// TwinCAT 3 PLC project hxr_jjslit_motion
// ProgramVersion: 3.1.4022.7
// libraries:
//   lcls-twincat-motion, * (SLAC)
//   Tc2_Standard, * (Beckhoff Automation GmbH)
//   Tc2_System, * (Beckhoff Automation GmbH)
//   Tc3_Module, * (Beckhoff Automation GmbH)
// project tree:
//   / PlcTask.TcTTO (not stored)
//   POUs/ Main.TcPOU
// real-time tasks:
//   TASK PlcTask: cycle T#10ms, priority 20, ADS port 350
// motion (NC):
//   TASK NC-Task 1 SAF: cycle T#2ms, priority 4, ADS port 501
//   TASK NC-Task 1 SVB: cycle T#10ms, priority 8, ADS port 511
//   AXIS VonHamosY (id 1)
//     Dynamic: AccelerationMaximum=30, DecelerationMaximum=30, Acceleration=14.9254, Deceleration=14.9254, Jerk=44.5534, DelayTime=0.008
//     Velo: RefSearch=0.1, RefSync=0.1, SlowManual=0.1, FastManual=0.2, Maximum=1.5
//     OtherSettings: AllowMotionCmdToSlave=true, PulseDistancePos=0.5, PulseDistanceNeg=0.5
//     encoder EncType=4
//       EncPara: ScaleFactorNumerator=1.5625e-05, Inverse=true, MaxCount=#x0000ffff
//         SoftEndMaxControl: Enable=true, Range=25
//         Inc: RefSoftSyncMask=#x0000ffff
//     drive DrvType=24
//       DrvPara: Inverse=true
//         Analog: VeloReferenz=2, ScaleFactorActTorque=0.1
//         TimeComp: TaskDelayCycles=1
//     controller CtrType=1
//       CtrPara: PriorControlFactor=1
//         PosDiffControl: Range=1
//         Observer: BandWidth=20
//   AXIS Axis 2 (Spare) (id 2)
//     OtherSettings: AllowMotionCmdToSlave=true
//     encoder EncType=4
//       EncPara: MaxCount=#x0000ffff
//         Inc: RefSoftSyncMask=#x0000ffff
//     drive DrvType=24
//       Analog: ScaleFactorActTorque=0.1
//       TimeComp: TaskDelayCycles=1
//     controller CtrType=1
//       CtrPara: PriorControlFactor=1
//         Observer: BandWidth=20
//   AXIS Axis 3 (Spare) (id 3)
//     OtherSettings: AllowMotionCmdToSlave=true
//     encoder EncType=4
//       EncPara: MaxCount=#x0000ffff
//         Inc: RefSoftSyncMask=#x0000ffff
//     drive DrvType=24
//       Analog: ScaleFactorActTorque=0.1
//       TimeComp: TaskDelayCycles=1
//     controller CtrType=1
//       CtrPara: PriorControlFactor=1
//         Observer: BandWidth=20
//   AXIS Axis 4 (Spare) (id 4)
//     OtherSettings: AllowMotionCmdToSlave=true
//     encoder EncType=4
//       EncPara: MaxCount=#x0000ffff
//         Inc: RefSoftSyncMask=#x0000ffff
//     drive DrvType=24
//       Analog: ScaleFactorActTorque=0.1
//       TimeComp: TaskDelayCycles=1
//     controller CtrType=1
//       CtrPara: PriorControlFactor=1
//         Observer: BandWidth=20
// I/O:
//   DEVICE Device 1 (EtherCAT), AmsNetId 5.63.55.4.2.1
//     VonHamos_EK1200_E0
// variable links:
//   (this object) <-> Device 1 (EtherCAT)/VonHamos_EK1200_E0/VonHamos_EL7041_E1
//     Drive/Inputs/In/nState1 @bit 3 <-> STM Status/Status/Error
//     Drive/Inputs/In/nState1 @bit 5 <-> STM Status/Status/Moving negative
//     Drive/Inputs/In/nState1 @bit 4 <-> STM Status/Status/Moving positive
//     Drive/Inputs/In/nState1 @bit 1 <-> STM Status/Status/Ready
//     Drive/Inputs/In/nState1 <-> STM Status/Status/Ready to enable
//     Drive/Inputs/In/nState1 @bit 6 <-> STM Status/Status/Torque reduced
//     Drive/Inputs/In/nState1 @bit 2 <-> STM Status/Status/Warning
//     Drive/Inputs/In/nState2 @bit 3 <-> STM Status/Status/Digital input 1
//     Drive/Inputs/In/nState2 @bit 4 <-> STM Status/Status/Digital input 2
//     Drive/Inputs/In/nState2 @bit 5 <-> STM Status/Status/Sync error
//     Drive/Inputs/In/nState2 @bit 7 <-> STM Status/Status/TxPDO Toggle
//     Drive/Inputs/In/nState4 @bit 1 <-> WcState/InputToggle
//     Drive/Inputs/In/nState4 <-> WcState/WcState
//     Drive/Outputs/Out/nCtrl1 <-> STM Control/Control/Enable
//     Drive/Outputs/Out/nCtrl1 @bit 2 <-> STM Control/Control/Reduce torque
//     Drive/Outputs/Out/nCtrl1 @bit 1 <-> STM Control/Control/Reset
//     Drive/Outputs/Out/nDataOut2[0] <-> STM Velocity/Velocity
//     Enc/Inputs/In/nDataIn1[0] <-> ENC Status compact/Counter value
//     Enc/Inputs/In/nDataIn2[0] <-> ENC Status compact/Latch value
//     Enc/Inputs/In/nState1 @bit 4 <-> ENC Status compact/Status/Counter overflow
//     Enc/Inputs/In/nState1 @bit 3 <-> ENC Status compact/Status/Counter underflow
//     Enc/Inputs/In/nState1 @bit 7 <-> ENC Status compact/Status/Extrapolation stall
//     Enc/Inputs/In/nState1 <-> ENC Status compact/Status/Latch C valid
//     Enc/Inputs/In/nState1 @bit 1 <-> ENC Status compact/Status/Latch extern valid
//     Enc/Inputs/In/nState1 @bit 2 <-> ENC Status compact/Status/Set counter done
//     Enc/Inputs/In/nState2 @bit 4 <-> ENC Status compact/Status/Status of extern latch
//     Enc/Inputs/In/nState2 <-> ENC Status compact/Status/Status of input A
//     Enc/Inputs/In/nState2 @bit 1 <-> ENC Status compact/Status/Status of input B
//     Enc/Inputs/In/nState2 @bit 2 <-> ENC Status compact/Status/Status of input C
//     Enc/Inputs/In/nState2 @bit 5 <-> ENC Status compact/Status/Sync error
//     Enc/Inputs/In/nState2 @bit 7 <-> ENC Status compact/Status/TxPDO Toggle
//     Enc/Inputs/In/nState4 @bit 1 <-> WcState/InputToggle
//     Enc/Inputs/In/nState4 <-> WcState/WcState
//     Enc/Outputs/Out/nCtrl1 <-> ENC Control compact/Control/Enable latch C
//     Enc/Outputs/Out/nCtrl1 @bit 3 <-> ENC Control compact/Control/Enable latch extern on negative edge
//     Enc/Outputs/Out/nCtrl1 @bit 1 <-> ENC Control compact/Control/Enable latch extern on positive edge
//     Enc/Outputs/Out/nCtrl1 @bit 2 <-> ENC Control compact/Control/Set counter
//     Enc/Outputs/Out/nDataOut1[0] <-> ENC Control compact/Set counter value
//   (this object) <-> Device 1 (EtherCAT)/VonHamos_EK1200_E0/VonHamos_EL7041_E3
//     Drive/Inputs/In/nState1 @bit 3 <-> STM Status/Status/Error
//     Drive/Inputs/In/nState1 @bit 5 <-> STM Status/Status/Moving negative
//     Drive/Inputs/In/nState1 @bit 4 <-> STM Status/Status/Moving positive
//     Drive/Inputs/In/nState1 @bit 1 <-> STM Status/Status/Ready
//     Drive/Inputs/In/nState1 <-> STM Status/Status/Ready to enable
//     Drive/Inputs/In/nState1 @bit 6 <-> STM Status/Status/Torque reduced
//     Drive/Inputs/In/nState1 @bit 2 <-> STM Status/Status/Warning
//     Drive/Inputs/In/nState2 @bit 3 <-> STM Status/Status/Digital input 1
//     Drive/Inputs/In/nState2 @bit 4 <-> STM Status/Status/Digital input 2
//     Drive/Inputs/In/nState2 @bit 5 <-> STM Status/Status/Sync error
//     Drive/Inputs/In/nState2 @bit 7 <-> STM Status/Status/TxPDO Toggle
//     Drive/Inputs/In/nState4 @bit 1 <-> WcState/InputToggle
//     Drive/Inputs/In/nState4 <-> WcState/WcState
//     Drive/Outputs/Out/nCtrl1 <-> STM Control/Control/Enable
//     Drive/Outputs/Out/nCtrl1 @bit 2 <-> STM Control/Control/Reduce torque
//     Drive/Outputs/Out/nCtrl1 @bit 1 <-> STM Control/Control/Reset
//     Drive/Outputs/Out/nDataOut2[0] <-> STM Velocity/Velocity
//     Enc/Inputs/In/nDataIn1[0] <-> ENC Status compact/Counter value
//     Enc/Inputs/In/nDataIn2[0] <-> ENC Status compact/Latch value
//     Enc/Inputs/In/nState1 @bit 4 <-> ENC Status compact/Status/Counter overflow
//     Enc/Inputs/In/nState1 @bit 3 <-> ENC Status compact/Status/Counter underflow
//     Enc/Inputs/In/nState1 @bit 7 <-> ENC Status compact/Status/Extrapolation stall
//     Enc/Inputs/In/nState1 <-> ENC Status compact/Status/Latch C valid
//     Enc/Inputs/In/nState1 @bit 1 <-> ENC Status compact/Status/Latch extern valid
//     Enc/Inputs/In/nState1 @bit 2 <-> ENC Status compact/Status/Set counter done
//     Enc/Inputs/In/nState2 @bit 4 <-> ENC Status compact/Status/Status of extern latch
//     Enc/Inputs/In/nState2 <-> ENC Status compact/Status/Status of input A
//     Enc/Inputs/In/nState2 @bit 1 <-> ENC Status compact/Status/Status of input B
//     Enc/Inputs/In/nState2 @bit 2 <-> ENC Status compact/Status/Status of input C
//     Enc/Inputs/In/nState2 @bit 5 <-> ENC Status compact/Status/Sync error
//     Enc/Inputs/In/nState2 @bit 7 <-> ENC Status compact/Status/TxPDO Toggle
//     Enc/Inputs/In/nState4 @bit 1 <-> WcState/InputToggle
//     Enc/Inputs/In/nState4 <-> WcState/WcState
//     Enc/Outputs/Out/nCtrl1 <-> ENC Control compact/Control/Enable latch C
//     Enc/Outputs/Out/nCtrl1 @bit 3 <-> ENC Control compact/Control/Enable latch extern on negative edge
//     Enc/Outputs/Out/nCtrl1 @bit 1 <-> ENC Control compact/Control/Enable latch extern on positive edge
//     Enc/Outputs/Out/nCtrl1 @bit 2 <-> ENC Control compact/Control/Set counter
//     Enc/Outputs/Out/nDataOut1[0] <-> ENC Control compact/Set counter value
//   (this object) <-> Device 1 (EtherCAT)/VonHamos_EK1200_E0/VonHamos_EL7041_E4
//     Drive/Inputs/In/nState1 @bit 3 <-> STM Status/Status/Error
//     Drive/Inputs/In/nState1 @bit 5 <-> STM Status/Status/Moving negative
//     Drive/Inputs/In/nState1 @bit 4 <-> STM Status/Status/Moving positive
//     Drive/Inputs/In/nState1 @bit 1 <-> STM Status/Status/Ready
//     Drive/Inputs/In/nState1 <-> STM Status/Status/Ready to enable
//     Drive/Inputs/In/nState1 @bit 6 <-> STM Status/Status/Torque reduced
//     Drive/Inputs/In/nState1 @bit 2 <-> STM Status/Status/Warning
//     Drive/Inputs/In/nState2 @bit 3 <-> STM Status/Status/Digital input 1
//     Drive/Inputs/In/nState2 @bit 4 <-> STM Status/Status/Digital input 2
//     Drive/Inputs/In/nState2 @bit 5 <-> STM Status/Status/Sync error
//     Drive/Inputs/In/nState2 @bit 7 <-> STM Status/Status/TxPDO Toggle
//     Drive/Inputs/In/nState4 @bit 1 <-> WcState/InputToggle
//     Drive/Inputs/In/nState4 <-> WcState/WcState
//     Drive/Outputs/Out/nCtrl1 <-> STM Control/Control/Enable
//     Drive/Outputs/Out/nCtrl1 @bit 2 <-> STM Control/Control/Reduce torque
//     Drive/Outputs/Out/nCtrl1 @bit 1 <-> STM Control/Control/Reset
//     Drive/Outputs/Out/nDataOut2[0] <-> STM Velocity/Velocity
//     Enc/Inputs/In/nDataIn1[0] <-> ENC Status compact/Counter value
//     Enc/Inputs/In/nDataIn2[0] <-> ENC Status compact/Latch value
//     Enc/Inputs/In/nState1 @bit 4 <-> ENC Status compact/Status/Counter overflow
//     Enc/Inputs/In/nState1 @bit 3 <-> ENC Status compact/Status/Counter underflow
//     Enc/Inputs/In/nState1 @bit 7 <-> ENC Status compact/Status/Extrapolation stall
//     Enc/Inputs/In/nState1 <-> ENC Status compact/Status/Latch C valid
//     Enc/Inputs/In/nState1 @bit 1 <-> ENC Status compact/Status/Latch extern valid
//     Enc/Inputs/In/nState1 @bit 2 <-> ENC Status compact/Status/Set counter done
//     Enc/Inputs/In/nState2 @bit 4 <-> ENC Status compact/Status/Status of extern latch
//     Enc/Inputs/In/nState2 <-> ENC Status compact/Status/Status of input A
//     Enc/Inputs/In/nState2 @bit 1 <-> ENC Status compact/Status/Status of input B
//     Enc/Inputs/In/nState2 @bit 2 <-> ENC Status compact/Status/Status of input C
//     Enc/Inputs/In/nState2 @bit 5 <-> ENC Status compact/Status/Sync error
//     Enc/Inputs/In/nState2 @bit 7 <-> ENC Status compact/Status/TxPDO Toggle
//     Enc/Inputs/In/nState4 @bit 1 <-> WcState/InputToggle
//     Enc/Inputs/In/nState4 <-> WcState/WcState
//     Enc/Outputs/Out/nCtrl1 <-> ENC Control compact/Control/Enable latch C
//     Enc/Outputs/Out/nCtrl1 @bit 3 <-> ENC Control compact/Control/Enable latch extern on negative edge
//     Enc/Outputs/Out/nCtrl1 @bit 1 <-> ENC Control compact/Control/Enable latch extern on positive edge
//     Enc/Outputs/Out/nCtrl1 @bit 2 <-> ENC Control compact/Control/Set counter
//     Enc/Outputs/Out/nDataOut1[0] <-> ENC Control compact/Set counter value
//   (this object) <-> Device 1 (EtherCAT)/VonHamos_EK1200_E0/VonHamos_EL7041_E6
//     Drive/Inputs/In/nState1 @bit 3 <-> STM Status/Status/Error
//     Drive/Inputs/In/nState1 @bit 5 <-> STM Status/Status/Moving negative
//     Drive/Inputs/In/nState1 @bit 4 <-> STM Status/Status/Moving positive
//     Drive/Inputs/In/nState1 @bit 1 <-> STM Status/Status/Ready
//     Drive/Inputs/In/nState1 <-> STM Status/Status/Ready to enable
//     Drive/Inputs/In/nState1 @bit 6 <-> STM Status/Status/Torque reduced
//     Drive/Inputs/In/nState1 @bit 2 <-> STM Status/Status/Warning
//     Drive/Inputs/In/nState2 @bit 3 <-> STM Status/Status/Digital input 1
//     Drive/Inputs/In/nState2 @bit 4 <-> STM Status/Status/Digital input 2
//     Drive/Inputs/In/nState2 @bit 5 <-> STM Status/Status/Sync error
//     Drive/Inputs/In/nState2 @bit 7 <-> STM Status/Status/TxPDO Toggle
//     Drive/Inputs/In/nState4 @bit 1 <-> WcState/InputToggle
//     Drive/Inputs/In/nState4 <-> WcState/WcState
//     Drive/Outputs/Out/nCtrl1 <-> STM Control/Control/Enable
//     Drive/Outputs/Out/nCtrl1 @bit 2 <-> STM Control/Control/Reduce torque
//     Drive/Outputs/Out/nCtrl1 @bit 1 <-> STM Control/Control/Reset
//     Drive/Outputs/Out/nDataOut2[0] <-> STM Velocity/Velocity
//     Enc/Inputs/In/nDataIn1[0] <-> ENC Status compact/Counter value
//     Enc/Inputs/In/nDataIn2[0] <-> ENC Status compact/Latch value
//     Enc/Inputs/In/nState1 @bit 4 <-> ENC Status compact/Status/Counter overflow
//     Enc/Inputs/In/nState1 @bit 3 <-> ENC Status compact/Status/Counter underflow
//     Enc/Inputs/In/nState1 @bit 7 <-> ENC Status compact/Status/Extrapolation stall
//     Enc/Inputs/In/nState1 <-> ENC Status compact/Status/Latch C valid
//     Enc/Inputs/In/nState1 @bit 1 <-> ENC Status compact/Status/Latch extern valid
//     Enc/Inputs/In/nState1 @bit 2 <-> ENC Status compact/Status/Set counter done
//     Enc/Inputs/In/nState2 @bit 4 <-> ENC Status compact/Status/Status of extern latch
//     Enc/Inputs/In/nState2 <-> ENC Status compact/Status/Status of input A
//     Enc/Inputs/In/nState2 @bit 1 <-> ENC Status compact/Status/Status of input B
//     Enc/Inputs/In/nState2 @bit 2 <-> ENC Status compact/Status/Status of input C
//     Enc/Inputs/In/nState2 @bit 5 <-> ENC Status compact/Status/Sync error
//     Enc/Inputs/In/nState2 @bit 7 <-> ENC Status compact/Status/TxPDO Toggle
//     Enc/Inputs/In/nState4 @bit 1 <-> WcState/InputToggle
//     Enc/Inputs/In/nState4 <-> WcState/WcState
//     Enc/Outputs/Out/nCtrl1 <-> ENC Control compact/Control/Enable latch C
//     Enc/Outputs/Out/nCtrl1 @bit 3 <-> ENC Control compact/Control/Enable latch extern on negative edge
//     Enc/Outputs/Out/nCtrl1 @bit 1 <-> ENC Control compact/Control/Enable latch extern on positive edge
//     Enc/Outputs/Out/nCtrl1 @bit 2 <-> ENC Control compact/Control/Set counter
//     Enc/Outputs/Out/nDataOut1[0] <-> ENC Control compact/Set counter value
//   hxr_jjslit_motion Instance <-> Device 1 (EtherCAT)/VonHamos_EK1200_E0/VonHamos_EL1084_E2
//     PlcTask Inputs/Main.M1.bHome <-> Channel 3/Input
//     PlcTask Inputs/Main.M1.bLimitBackwardEnable <-> Channel 2/Input
//     PlcTask Inputs/Main.M1.bLimitForwardEnable <-> Channel 1/Input
//   hxr_jjslit_motion Instance <-> Device 1 (EtherCAT)/VonHamos_EK1200_E0/VonHamos_EL2004_E7
//     PlcTask Outputs/Main.M1.bBrakeRelease <-> Channel 1/Output
//   hxr_jjslit_motion Instance <-> NC-Task 1 SAF/Axes/JJ_1_V_Gap
//     PlcTask Inputs/Main.M1.Axis.NcToPlc <-> Outputs/ToPlc
//     PlcTask Outputs/Main.M1.Axis.PlcToNc <-> Inputs/FromPlc

// ---- POUs/Main.TcPOU
PROGRAM Main
VAR
	// Motors
	{attribute 'TcLinkTo' := '.bLimitForwardEnable	:=TIIB[JJ_1_V_Gap_EL7037]^Channel 1^Input;
                              .bLimitBackwardEnable	:=TIIB[JJ_1_V_Gap_EL7037]^Channel 2^Input;
	{attribute 'pytmc' := '
		pv: XPP:JJAT:MMS:01
	'}
	M1 : DUT_MotionStage := (bPowerSelf:=True); // JJ_1_Vertical_Gap

	fbMotionStageM1 : FB_MotionStage;
	
	
	{attribute 'TcLinkTo' := '.bLimitForwardEnable	:=TIIB[JJ_1_V_Offset_EL7037]^Channel 1^Input;
                              .bLimitBackwardEnable	:=TIIB[JJ_1_V_Offset_EL7037]^Channel 2^Input;
	{attribute 'pytmc' := '
		pv: XPP:JJAT:MMS:02
	'}
	M2 : DUT_MotionStage := (bPowerSelf:=True); // JJ_1_Vertical_Offset

	fbMotionStageM2 : FB_MotionStage;
	
	{attribute 'TcLinkTo' := '.bLimitForwardEnable	:=TIIB[JJ_1_H_Gap_EL7037]^Channel 1^Input;
                              .bLimitBackwardEnable	:=TIIB[JJ_1_H_Gap_EL7037]^Channel 2^Input;
	{attribute 'pytmc' := '
		pv: XPP:JJAT:MMS:03
	'}
	M3 : DUT_MotionStage := (bPowerSelf:=True); // JJ_1_Horizontal_Gap

	fbMotionStageM3 : FB_MotionStage;
	
	{attribute 'TcLinkTo' := '.bLimitForwardEnable	:=TIIB[JJ_1_H_Offset_EL7037]^Channel 1^Input;
                              .bLimitBackwardEnable	:=TIIB[JJ_1_H_Offset_EL7037]^Channel 2^Input;
	{attribute 'pytmc' := '
		pv: XPP:JJAT:MMS:04
	'}
	M4 : DUT_MotionStage := (bPowerSelf:=True); // JJ_1_Horizontal_Offset

	fbMotionStageM4 : FB_MotionStage;
	
	{attribute 'TcLinkTo' := '.bLimitForwardEnable	:=TIIB[JJ_2_V_Gap_EL7037]^Channel 1^Input;
                              .bLimitBackwardEnable	:=TIIB[JJ_2_V_Gap_EL7037]^Channel 2^Input;
	{attribute 'pytmc' := '
		pv: XPP:JJAT:MMS:05
	'}
	M5 : DUT_MotionStage := (bPowerSelf:=True); // JJ_2_Vertical_Gap

	fbMotionStageM5 : FB_MotionStage;
	
	{attribute 'TcLinkTo' := '.bLimitForwardEnable	:=TIIB[JJ_2_V_Offset_EL7037]^Channel 1^Input;
                              .bLimitBackwardEnable	:=TIIB[JJ_2_V_Offset_EL7037]^Channel 2^Input;
	{attribute 'pytmc' := '
		pv: XPP:JJAT:MMS:06
	'}
	M6 : DUT_MotionStage := (bPowerSelf:=True); // JJ_2_Vertical_Offset

	fbMotionStageM6 : FB_MotionStage;
	
	{attribute 'TcLinkTo' := '.bLimitForwardEnable	:=TIIB[JJ_2_H_Gap_EL7037]^Channel 1^Input;
                              .bLimitBackwardEnable	:=TIIB[JJ_2_H_Gap_EL7037]^Channel 2^Input;
	{attribute 'pytmc' := '
		pv: XPP:JJAT:MMS:07
	'}
	M7 : DUT_MotionStage := (bPowerSelf:=True); // JJ_2_Horizontal_Gap

	fbMotionStageM7 : FB_MotionStage;
	
	{attribute 'TcLinkTo' := '.bLimitForwardEnable	:=TIIB[JJ_2_H_Offset_EL7037]^Channel 1^Input;
                              .bLimitBackwardEnable	:=TIIB[JJ_2_V_Offset_EL7037]^Channel 2^Input;
	{attribute 'pytmc' := '
		pv: XPP:JJAT:MMS:08
	'}
	M8 : DUT_MotionStage := (bPowerSelf:=True); // JJ_2_Horizontal_Offset

	fbMotionStageM8 : FB_MotionStage;
	
	{attribute 'TcLinkTo' := '.bLimitForwardEnable	:=TIIB[JJ_3_V_Gap_EL7037]^Channel 1^Input;
                              .bLimitBackwardEnable	:=TIIB[JJ_3_V_Gap_EL7037]^Channel 2^Input;
	{attribute 'pytmc' := '
		pv: XPP:JJAT:MMS:09
	'}
	M9 : DUT_MotionStage := (bPowerSelf:=True); // JJ_3_Vertical_Gap

	fbMotionStageM9 : FB_MotionStage;
	
	{attribute 'TcLinkTo' := '.bLimitForwardEnable	:=TIIB[JJ_3_V_Offset_EL7037]^Channel 1^Input;
                              .bLimitBackwardEnable	:=TIIB[JJ_3_V_Offset_EL7037]^Channel 2^Input;
	{attribute 'pytmc' := '
		pv: XPP:JJAT:MMS:10
	'}
	M10 : DUT_MotionStage := (bPowerSelf:=True); // JJ_3_Vertical_Offset

	fbMotionStageM10 : FB_MotionStage;
	
	{attribute 'TcLinkTo' := '.bLimitForwardEnable	:=TIIB[JJ_3_H_Gap_EL7037]^Channel 1^Input;
                              .bLimitBackwardEnable	:=TIIB[JJ_3_H_Gap_EL7037]^Channel 2^Input;
	{attribute 'pytmc' := '
		pv: XPP:JJAT:MMS:11
	'}
	M11 : DUT_MotionStage := (bPowerSelf:=True); // JJ_3_Horizontal_Gap

	fbMotionStageM11 : FB_MotionStage;
	
	{attribute 'TcLinkTo' := '.bLimitForwardEnable	:=TIIB[JJ_3_H_Offset_EL7037]^Channel 1^Input;
                              .bLimitBackwardEnable	:=TIIB[JJ_3_H_Offset_EL7037]^Channel 2^Input;
	{attribute 'pytmc' := '
		pv: XPP:JJAT:MMS:12
	'}
	M12 : DUT_MotionStage := (bPowerSelf:=True); // JJ_3_Horizontal_Offset

	fbMotionStageM12 : FB_MotionStage;
	
	{attribute 'TcLinkTo' := '.bLimitForwardEnable	:=TIIB[JJ_4_V_Gap_EL7037]^Channel 1^Input;
                              .bLimitBackwardEnable	:=TIIB[JJ_4_V_Gap_EL7037]^Channel 2^Input;
	{attribute 'pytmc' := '
		pv: XPP:JJAT:MMS:13
	'}
	M13 : DUT_MotionStage := (bPowerSelf:=True); // JJ_4_Vertical_Gap

	fbMotionStageM13 : FB_MotionStage;
	
	{attribute 'TcLinkTo' := '.bLimitForwardEnable	:=TIIB[JJ_4_V_Offset_EL7037]^Channel 1^Input;
                              .bLimitBackwardEnable	:=TIIB[JJ_4_V_Offset_EL7037]^Channel 2^Input;
	{attribute 'pytmc' := '
		pv: XPP:JJAT:MMS:14
	'}
	M14 : DUT_MotionStage := (bPowerSelf:=True); // JJ_4_Vertical_Offset

	fbMotionStageM14 : FB_MotionStage;
	
	{attribute 'TcLinkTo' := '.bLimitForwardEnable	:=TIIB[JJ_4_H_Gap_EL7037]^Channel 1^Input;
                              .bLimitBackwardEnable	:=TIIB[JJ_4_H_Gap_EL7037]^Channel 2^Input;
	{attribute 'pytmc' := '
		pv: XPP:JJAT:MMS:15
	'}
	M15 : DUT_MotionStage := (bPowerSelf:=True); // JJ_4_Horizontal_Gap

	fbMotionStageM15 : FB_MotionStage;
	
	{attribute 'TcLinkTo' := '.bLimitForwardEnable	:=TIIB[JJ_4_H_Offset_EL7037]^Channel 1^Input;
                              .bLimitBackwardEnable	:=TIIB[JJ_4_H_Offset_EL7037]^Channel 2^Input;
	{attribute 'pytmc' := '
		pv: XPP:JJAT:MMS:16
	'}
	M16 : DUT_MotionStage := (bPowerSelf:=True); // JJ_4_Horizontal_Offset

	fbMotionStageM16 : FB_MotionStage;
END_VAR

// Hardware Enable
M1.bHardwareEnable := TRUE;
fbMotionStageM1(stMotionStage:=M1);

M2.bHardwareEnable := TRUE;
fbMotionStageM2(stMotionStage:=M2);

M3.bHardwareEnable := TRUE;
fbMotionStageM1(stMotionStage:=M3);

M4.bHardwareEnable := TRUE;
fbMotionStageM1(stMotionStage:=M4);

M5.bHardwareEnable := TRUE;
fbMotionStageM5(stMotionStage:=M5);

M6.bHardwareEnable := TRUE;
fbMotionStageM6(stMotionStage:=M6);

M3.bHardwareEnable := TRUE;
fbMotionStageM1(stMotionStage:=M3);

M7.bHardwareEnable := TRUE;
fbMotionStageM7(stMotionStage:=M7);

M8.bHardwareEnable := TRUE;
fbMotionStageM8(stMotionStage:=M8);

M9.bHardwareEnable := TRUE;
fbMotionStageM9(stMotionStage:=M9);

M10.bHardwareEnable := TRUE;
fbMotionStageM10(stMotionStage:=M10);

M11.bHardwareEnable := TRUE;
fbMotionStageM11(stMotionStage:=M11);

M12.bHardwareEnable := TRUE;
fbMotionStageM12(stMotionStage:=M12);

M13.bHardwareEnable := TRUE;
fbMotionStageM13(stMotionStage:=M13);

M14.bHardwareEnable := TRUE;
fbMotionStageM14(stMotionStage:=M14);

M15.bHardwareEnable := TRUE;
fbMotionStageM15(stMotionStage:=M15);

M1.bHardwareEnable := TRUE;
fbMotionStageM1(stMotionStage:=M1);

M2.bHardwareEnable := TRUE;
fbMotionStageM2(stMotionStage:=M2);

M3.bHardwareEnable := TRUE;
fbMotionStageM1(stMotionStage:=M3);

M16.bHardwareEnable := TRUE;
fbMotionStageM1(stMotionStage:=M16);

END_PROGRAM
